// TwinCAT 3 PLC project Blink
// ProgramVersion: 3.1.4022.4
// libraries:
//   Tc2_Standard, * (Beckhoff Automation GmbH)
//   Tc2_System, * (Beckhoff Automation GmbH)
//   Tc3_Module, * (Beckhoff Automation GmbH)
// project tree:
//   DUTs/ S_PulseOutput.TcDUT, S_PulseOutputV2.TcDUT, S_State.TcDUT
//   FBs/ FB_Blink.TcPOU, FB_Blinking.TcPOU, FB_Generator.TcPOU, FB_GeneratorEx.TcPOU
//   GVLs/ GVL_General.TcGVL
//   Interface/ IGenerator.TcIO
//   / PlcTask.TcTTO
//   POUs/ MAIN.TcPOU, PulsGenerator.TcPOU, PulsGeneratorV2.TcPOU
// real-time tasks:
//   TASK PlcTask: cycle T#10ms, priority 20, ADS port 350

CONFIGURATION Blink
    RESOURCE PLC ON TwinCAT3
        TASK PlcTask(INTERVAL := T#10ms, PRIORITY := 20);
        PROGRAM MAIN WITH PlcTask : MAIN;
    END_RESOURCE
END_CONFIGURATION

// ---- DUTs/S_PulseOutput.TcDUT
TYPE S_PulseOutput :
STRUCT
	Pulse100ms		:BOOL;
	Pulse200ms		:BOOL;
	Pulse500ms		:BOOL;
	Pulse800ms		:BOOL;
	Pulse1s			:BOOL;
	Pulse2s			:BOOL;	
END_STRUCT
END_TYPE

// ---- DUTs/S_PulseOutputV2.TcDUT
TYPE S_PulseOutputV2 :
STRUCT
	t100ms				: BOOL;
	t200ms				: BOOL;
	t250ms				: BOOL;
	t500ms				: BOOL;
	t750ms				: BOOL;
	t800ms				: BOOL;

	t1s					: BOOL;
	t2s					: BOOL;
END_STRUCT
END_TYPE

// ---- DUTs/S_State.TcDUT
TYPE S_State :
STRUCT
	pulse			:S_PulseOutputV2;
END_STRUCT
END_TYPE

// ---- GVLs/GVL_General.TcGVL
{attribute 'qualified_only'}
VAR_GLOBAL
	PulseOutput		:S_PulseOutput;
	state			:S_State;
END_VAR

// ---- Interface/IGenerator.TcIO
INTERFACE IGenerator

METHOD Flash : BOOL
VAR_INPUT
END_VAR
END_METHOD

PROPERTY P_tCycleTime : Time
GET
END_GET
SET
END_SET
END_PROPERTY

PROPERTY P_Vendor : string
GET
END_GET
END_PROPERTY

END_INTERFACE

// ---- POUs/MAIN.TcPOU
PROGRAM MAIN
VAR
	// Create by Huang Hansheng 2019.09.14
	//-------------------------------------------//
	fbGenerator			: FB_Generator;
	fbGeneratorEx		:FB_GeneratorEx;
	iGenerator			:IGenerator;
	bChange				:BOOL;
	_tCycleTime			:TIME:= T#2S;
	sVendor				:STRING;
	bOutput				:BOOL;
	//------------------------------------//
	
	fbBlink			:FB_Blink;
	bOutput2		:BOOL;
	//--------------------------------------//
	fbBlinking			:FB_Blinking;
	poutGreenLed		:POINTER TO BOOL;
	outGreenLed			AT %Q*:BOOL;	
	//--------------------------------------------//
	outRedLed			AT %Q*:BOOL;

	
	
END_VAR

//--------------------------------------------------------------------------//
	IF	bChange THEN 
		iGenerator := fbGenerator;
	ELSE
		iGenerator := fbGeneratorEx;
	END_IF
	
	iGenerator.P_tCycleTime :=  _tCycleTime;
	
	bOutput :=  iGenerator.Flash();
	
	sVendor := iGenerator.P_Vendor;
//-----------------------------------------------------------------//

fbBlink(msTime:= 300,sig=>bOutput2);

//------------------------------------------------------------//
	poutGreenLed := ADR(outGreenLed);
	fbBlinking(pVariable:=poutGreenLed , interval:= T#1S );
	
//------------------------------------------------------------//


	PulsGenerator();
	outRedLed := GVL_General.PulseOutput.Pulse1s;

	PulsGeneratorV2();

END_PROGRAM

// ---- FBs/FB_Generator.TcPOU
FUNCTION_BLOCK FB_Generator IMPLEMENTS IGenerator
VAR_INPUT
END_VAR
VAR_OUTPUT
END_VAR
VAR
	ton1		:TON;
	tCycleTime		:TIME;
	bBlink			:BOOL;
END_VAR

{warning 'add method implementation'}
METHOD Flash : BOOL
ton1(IN:=NOT ton1.Q, PT:= tCycleTime, Q=> , ET=> );

IF	ton1.Q THEN 
	bBlink := NOT bBlink;
END_IF

Flash	:= bBlink;
END_METHOD

{warning 'add property implementation'}
PROPERTY P_tCycleTime : TIME
GET
P_tCycleTime := tCycleTime;
END_GET
SET
tCycleTime := P_tCycleTime;
END_SET
END_PROPERTY

{warning 'add property implementation'}
PROPERTY P_Vendor : STRING
GET
P_Vendor := 'Google';
END_GET
END_PROPERTY

END_FUNCTION_BLOCK

// ---- FBs/FB_GeneratorEx.TcPOU
FUNCTION_BLOCK FB_GeneratorEx EXTENDS FB_Generator
VAR_INPUT
END_VAR
VAR_OUTPUT
END_VAR
VAR
END_VAR

{warning 'add method implementation'}
METHOD Flash : BOOL
ton1(IN:=NOT ton1.Q , PT:= tCycleTime, Q=> , ET=> );



// duty ratio 33% ON, 67% Off

Flash := ton1.ET < ton1.PT/3;
END_METHOD

PROPERTY P_tCycleTime : TIME
GET
P_tCycleTime := tCycleTime;
END_GET
SET
IF P_tCycleTime < T#50MS THEN 
	tCycleTime := T#50MS;
ELSIF P_tCycleTime > T#5S THEN 
	tCycleTime := T#5S;
ELSE
	tCycleTime := P_tCycleTime;	
END_IF
END_SET
END_PROPERTY

PROPERTY P_Vendor : STRING
GET
P_Vendor := CONCAT('MicroSoft',SUPER^.P_Vendor);
END_GET
END_PROPERTY

END_FUNCTION_BLOCK

// ---- FBs/FB_Blink.TcPOU
FUNCTION_BLOCK FB_Blink
VAR_INPUT
	msTime		:UDINT;	
END_VAR
VAR_OUTPUT
	sig		:BOOL;
END_VAR
VAR
	timeCounter		:UDINT;
	rtc				:GETCPUACCOUNT;
END_VAR

	
//
	rtc(cpuAccountDW=> );

	IF rtc.cpuAccountDW - timeCounter >= msTime*10000 THEN 
		sig := NOT sig;
		timeCounter := rtc.cpuAccountDW;
	END_IF

END_FUNCTION_BLOCK

// ---- FBs/FB_Blinking.TcPOU
FUNCTION_BLOCK FB_Blinking
VAR_INPUT
	pVariable		:POINTER TO BOOL;		//Address of variable to blink
	interval		:TIME;					//Blink interval
END_VAR
VAR_OUTPUT
END_VAR
VAR
	bState			:BOOL;
	tonTimer		:TON;
END_VAR

tonTimer(IN:=TRUE , PT:= interval);

IF tonTimer.Q THEN 
	bState := NOT bState;
	tonTimer(IN:=FALSE, PT:= interval);
END_IF

pVariable^ := bState;

END_FUNCTION_BLOCK

// ---- POUs/PulsGenerator.TcPOU
PROGRAM PulsGenerator
VAR
	fbBlinking,fbBlinking1,fbBlinking2,fbBlinking3,fbBlinking4,fbBlinking5		:FB_Blinking;
	pPulseOutput			:POINTER TO S_PulseOutput;
	
END_VAR

pPulseOutput := ADR(GVL_General.PulseOutput);


fbBlinking(pVariable:= ADR(pPulseOutput^.Pulse100ms) , interval:= T#100MS);

fbBlinking1(pVariable:= ADR(pPulseOutput^.Pulse1s) , interval:= T#1S);

fbBlinking2(pVariable:= ADR(pPulseOutput^.Pulse200ms) , interval:= T#200MS);

fbBlinking3(pVariable:= ADR(pPulseOutput^.Pulse2s) , interval:= T#2S);

fbBlinking4(pVariable:= ADR(pPulseOutput^.Pulse500ms) , interval:= T#500MS);

fbBlinking5(pVariable:= ADR(pPulseOutput^.Pulse800ms) , interval:= T#800MS);

END_PROGRAM

// ---- POUs/PulsGeneratorV2.TcPOU
PROGRAM PulsGeneratorV2
VAR
	timeCounter		:UDINT	:= 0;
	RTC		:GETCPUACCOUNT;
	tick50ms		:UDINT := 0;
	timeCounter2s		:UDINT:=0;
	tick2s				:UDINT:=1;
	tn					:DWORD;
	tx					:DWORD;
	init				:BOOL;
	
	timePlcMs			:UDINT;
	pulsChange			:BOOL:=FALSE;
	pulseChange: BOOL;
	//state: S_State;
	//pulse: INT;
	t100ms: BOOL;
	t200ms: BOOL;
	t250ms: BOOL;
	t500ms: BOOL;
	t750ms: BOOL;
	t800ms: BOOL;
	t1s: BOOL;
	t2s: BOOL;
END_VAR


timePlcMs	:= TIME_TO_UDINT(TIME());

(* reinit timeCounter if timePlcMs overflows *)
IF ( timePlcMs < timeCounter )
THEN
	timeCounter := 50 - (4294967295 - timeCounter);
END_IF

IF (timePlcMs - timeCounter) >= 50 THEN
	tick50ms := tick50ms + 1;
	timeCounter:=timePlcMs;
	pulseChange := TRUE;
END_IF

IF (pulseChange = TRUE)
THEN
	IF tick50ms MOD 2 = 0 THEN GVL_General.state.pulse.t100ms := NOT GVL_General.state.pulse.t100ms; END_IF
	IF tick50ms MOD 4 = 0 THEN GVL_General.state.pulse.t200ms := NOT GVL_General.state.pulse.t200ms; END_IF
	IF tick50ms MOD 5 = 0 THEN GVL_General.state.pulse.t250ms := NOT GVL_General.state.pulse.t250ms; END_IF
	IF tick50ms MOD 10 = 0 THEN GVL_General.state.pulse.t500ms := NOT GVL_General.state.pulse.t500ms; END_IF
	IF tick50ms MOD 15 = 0 THEN GVL_General.state.pulse.t750ms := NOT GVL_General.state.pulse.t750ms; END_IF
	IF tick50ms MOD 16 = 0 THEN GVL_General.state.pulse.t800ms := NOT GVL_General.state.pulse.t800ms; END_IF
	IF tick50ms MOD 20 = 0 THEN GVL_General.state.pulse.t1s := NOT GVL_General.state.pulse.t1s; END_IF
	IF tick50ms MOD 40 = 0 THEN GVL_General.state.pulse.t2s := NOT GVL_General.state.pulse.t2s; END_IF

	pulseChange := FALSE;

END_IF

END_PROGRAM
